// TIA Portal V20 export
DATA_BLOCK "Conveyor_C1_DB"   // DB3
// stored: InstanceOfName Conveyor_C1, InstanceOfType FB, Namespace Conveyor1
"Conveyor_C1"
   // VAR
   //    jogRight : Bool;
   // END_VAR
BEGIN
END_DATA_BLOCK
